(*********************************** G.D S.p.A. - Technical Department ***********************************
============= PROGRAM INFO ============
FOLDER:             TBD
MACHINES INVOLVED:  TBD 

============= DESCRIPTION =============

============= REVISIONS ===============
Date		Version	 	Author      	Description             
----------	-------		------------  	--------------------------------------------
2019/04/24 	0000.00	 	M.Grasso		Creation of the PRG

**********************************************************************************************************)
(*$R
	process_ref := prc;
$*)
PROGRAM csp_transfer_main_safety
VAR
	prc:					process;
	prc_path:				STRING;
END_VAR

_read_var_input();

_object_manager();

IF NOT objects_running()
THEN
	RETURN;	
END_IF

_read_process_image();

_mode_manager();

CASE process_get_mode(prc) of
	MODE_ABSENT,
	MODE_INACTIVE:
		RETURN;
	MODE_TEST:
		_handle_process_test();
END_CASE

_set_runtime_properties();

(********************************* BODY *********************************)

(************************************************************************)

_handle_messages();

_write_output();

ACTION _handle_messages:
;
END_ACTION

ACTION _handle_process_test:
;
END_ACTION

ACTION _mode_manager:
IF process_mode_req_is_pending(prc)
THEN
    process_apply_mode_req_first_step(prc);
    CASE process_get_mode(prc) OF
        MODE_TO_ABSENT:
			;
        MODE_TO_INACTIVE:
			;
        MODE_TO_TEST:
			;
        MODE_TO_OPERATIONAL:
			;
    END_CASE
    process_apply_mode_req_second_step(prc);
END_IF
END_ACTION

ACTION _object_manager:
IF objects_initialization()
THEN
	sub_process_init(
		object_name					:= 'csp_transfer_main_safety.prc', 
		process						:= csp_transfer_main.prc, 
		CONVERSION_this				:= prc);
		
	prc_path 						:= process_get_path(prc);
END_IF

IF objects_running()
THEN
	process_cycle(prc);
END_IF
END_ACTION

ACTION _read_process_image:
;
END_ACTION

ACTION _read_var_input:
;
END_ACTION

ACTION _set_runtime_properties:
;
END_ACTION

ACTION _write_output:
;
END_ACTION

END_PROGRAM

(* stored: Version 1.1.0.1, ProductVersion 3.1.4022.12
   POU csp_transfer_main_safety: Id {358aa4f7-b45c-4a45-8f47-88f38a9a9f40}, SpecialFunc None
   Action _handle_messages: Id {fdc33d09-5b73-48d1-a5d9-c6c458874974}
   Action _handle_process_test: Id {87f884ab-dfd9-4bfa-ad66-834387e4f371}
   Action _mode_manager: Id {741a80e9-6621-4561-8364-82ec56e4e881}
   Action _object_manager: Id {7d862e46-ac4e-4c43-8ee0-57106229a153}
   Action _read_process_image: Id {0fda3cf4-71b3-40fe-b09f-c5503f21bbe2}
   Action _read_var_input: Id {44f3dd7d-7085-42f2-a015-cf77a22f3c5c}
   Action _set_runtime_properties: Id {2f61023f-e657-43e7-92da-984c73ac6bd1}
   Action _write_output: Id {8486cfc7-fdb2-4924-83ff-f6aa7e5b7178} *)
